PROGRAM Faults
VAR
END_VAR

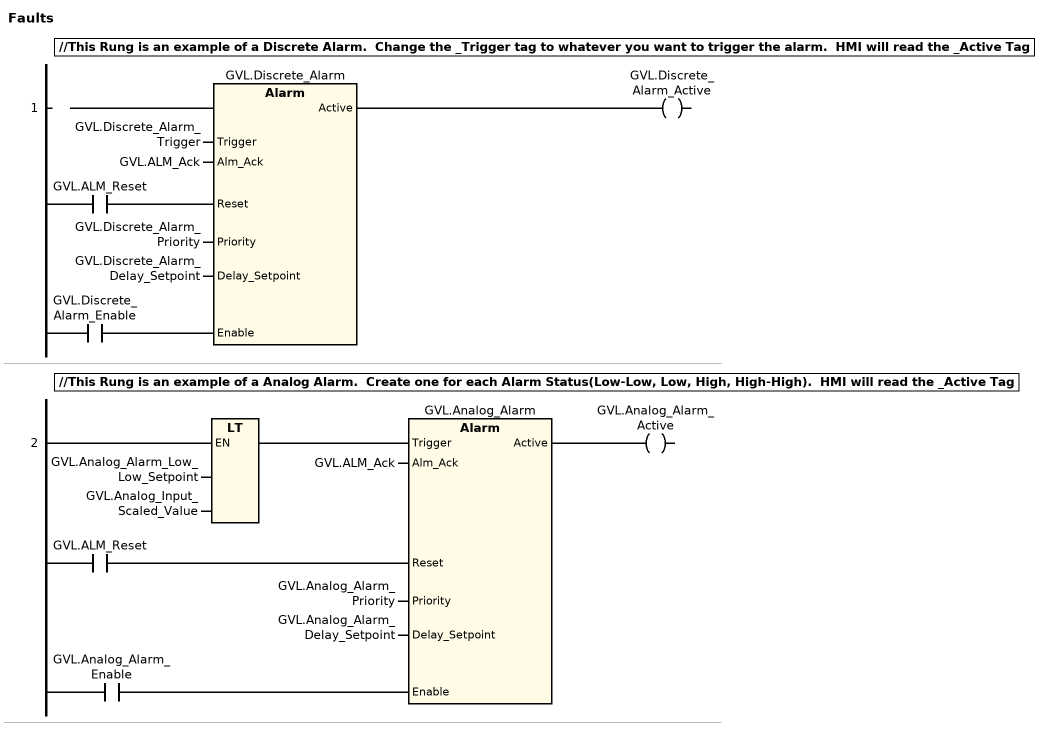
// NETWORK 1
// label: //This Rung is an example of a Discrete Alarm.  Change the _Trigger tag to whatever you want to trigger the alarm.  HMI will read the _Active Tag
GVL.Discrete_Alarm(
    Trigger := GVL.Discrete_Alarm_Trigger,
    Alm_Ack := GVL.ALM_Ack,
    Reset := GVL.ALM_Reset,
    Priority := GVL.Discrete_Alarm_Priority,
    Delay_Setpoint := GVL.Discrete_Alarm_Delay_Setpoint,
    Enable := GVL.Discrete_Alarm_Enable); // Alarm
GVL.Discrete_Alarm_Active := GVL.Discrete_Alarm.Active;

// NETWORK 2
// label: //This Rung is an example of a Analog Alarm.  Create one for each Alarm Status(Low-Low, Low, High, High-High).  HMI will read the _Active Tag
GVL.Analog_Alarm(
    Trigger := GVL.Analog_Alarm_Low_Low_Setpoint < GVL.Analog_Input_Scaled_Value,
    Alm_Ack := GVL.ALM_Ack,
    Reset := GVL.ALM_Reset,
    Priority := GVL.Analog_Alarm_Priority,
    Delay_Setpoint := GVL.Analog_Alarm_Delay_Setpoint,
    Enable := GVL.Analog_Alarm_Enable); // Alarm
GVL.Analog_Alarm_Active := GVL.Analog_Alarm.Active;

END_PROGRAM

(* stored: Version 1.1.0.1, ProductVersion 3.1.4024.12
   POU Faults: Id {6bd76c82-c4f2-4561-a2e5-6d6c31340040}, SpecialFunc None *)
